// TIA Portal V15.1 export
// export: Created 2024-06-21T08:40:55.5376107Z, ExportSetting WithDefaults, DisplayName Totally Integrated Automation Portal, DisplayVersion V15.1 Update 5, DisplayName TIA Portal Openness, DisplayVersion V15.1 Update 5, DisplayName SINAMICS Startdrive Advanced, DisplayVersion V15.1, DisplayName G130, G150, S120, S150, SINAMICS MV, S210, DisplayVersion V15.1, DisplayName G110M, G120, G120C, G120D, G120P, DisplayVersion V15.1, DisplayName STEP 7 Professional, DisplayVersion V15.1 Update 5, DisplayName STEP 7 Safety, DisplayVersion V15.1, DisplayName WinCC Professional, DisplayVersion V15.1 Update 5, DisplayName SIMATIC Visualization Architect, DisplayVersion V15.1
FUNCTION "LAlarmSummaryInit" : Void   // FC2538, FBD
TITLE = LAlarmSummary / LAlarmSummaryInit
{ S7_Optimized_Access := 'TRUE' }
VERSION : 0.1
// =============================================================================
// This module is used to sum all alarm's from all objects "FB&FC's" and the send it to LMode & LSystemVar-S71500
// =============================================================================
// =============================================================================
// FC to merge 1 Alarm UDT
// Shall be called in first network
// =============================================================================
// stored: AutoNumber false, IsIECCheckEnabled false, SetENOAutomatically False, UDAEnableTagReadback false
   VAR_IN_OUT
      IO_Alarm : "Alarm";   // Alarm UDT
   END_VAR
   VAR_TEMP   // added for the SCL form of the ladder/FBD networks
      _w1 : Bool;
   END_VAR
BEGIN

REGION Network 1: **** 1 - Inputs **** Init Alarm UDT Upper Level / **** 1 - Inputs **** Init Alarm UDT
   // Alarm / Alarm D / Init Alarm UDT
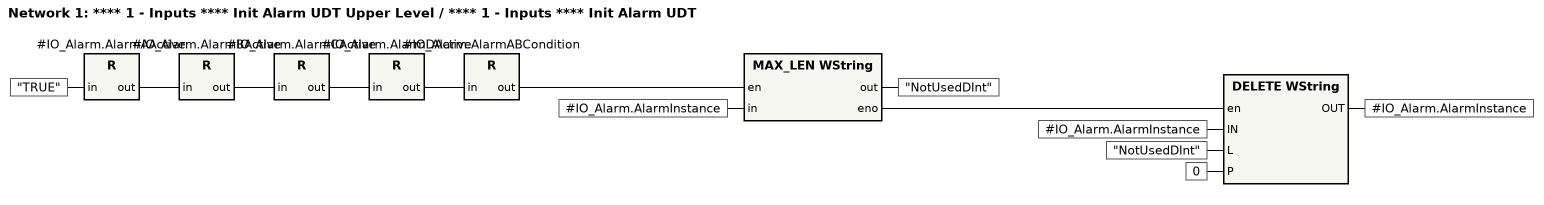
   // ENO of a box is taken as its EN; it also drops when the box reports an error
   IF "TRUE" THEN
       #IO_Alarm.AlarmAActive := FALSE;
       #IO_Alarm.AlarmBActive := FALSE;
       #IO_Alarm.AlarmCActive := FALSE;
       #IO_Alarm.AlarmDActive := FALSE;
       #IO_Alarm.AlarmABCondition := FALSE;
   END_IF;
   #_w1 := "TRUE";
   IF #_w1 THEN
       MAX_LEN(in := #IO_Alarm.AlarmInstance, out => "NotUsedDInt");
       DELETE(IN := #IO_Alarm.AlarmInstance, L := "NotUsedDInt", P := 0, OUT => #IO_Alarm.AlarmInstance);
   END_IF;
END_REGION
END_FUNCTION
